// TIA Portal project "Recepe" (V17)

(* hardware
DEVICE "HMI_1"  KTP400 Comfort
   slot 0: "HMI_1"  KTP400 Comfort  6AV2 124-2DC01-0AX0  17.0.0.0
   slot 1: "HMI_RT_1"  KTP400 Comfort  6AV2 124-2DC01-0AX0  17.0.0.0
   slot 5: "HMI_1.IE_CP_1"  PROFINET Interface  17.0.0.0
      slot 1: "PROFINET Interface_1"  PROFINET Interface
         slot 1: "Port_1"  Port
   slot 7: "HMI_1.MPI/DP_CP_1"  MPI/DP Interface  17.0.0.0
*)

(* ===== HMI "HMI_RT_1" =====
system functions are stored by id; their names below are inferred from use

recipe "Recipe_1": 

Template "Template_1" 480x272
   Button "Language" at 415,70 size 63x63; TextOff 'Language'; PictureOff "ToggleLanguage_KTP400_Comfort_TR"; PictureOn "ToggleLanguage_KTP400_Comfort_TR"
      on Release: function_fb9197e8(-1)
   Button "Log on" at 415,138 size 63x63; TextOff 'Log on'; PictureOff "Login_KTP400_Comfort_TR"; PictureOn "Login_KTP400_Comfort_TR"
      on Release: function_a2a04561()
   Button "Exit" at 415,207 size 63x63; TextOff 'Exit'; PictureOff "ExitRuntime_KTP400_Comfort_TR"; PictureOn "ExitRuntime_KTP400_Comfort_TR"
      on Release: StopRuntime(0)
   Button "Start screen" at 415,1 size 63x63; TextOff 'Start screen'; PictureOff "NavigateHome_KTP400_Comfort_TR"; PictureOn "NavigateHome_KTP400_Comfort_TR"
      on Release: ActivateScreen("Root screen", 0)
*)